% RSLogix 500 project Project2.RSS, saved by version 8.30.00.16 %
PROJECT "UNTITLED"    % processor: Bul.1763 MicroLogix 1100 Series B %

PROGRAM FILES
  LAD 2 "MAIN"  3 rungs
  LAD 3 "IO"  8 rungs
  LAD 4 "CONTROLS"  4 rungs

DATA FILES
  O0 OUTPUT  4 elements
  I1 INPUT  6 elements
  S2 STATUS  66 elements
  B3 BINARY  1 elements
  T4 TIMER  1 elements
  C5 COUNTER  1 elements
  R6 CONTROL  1 elements
  N7 INTEGER  1 elements
  F8 FLOAT  1 elements

LADDER 2 "MAIN"
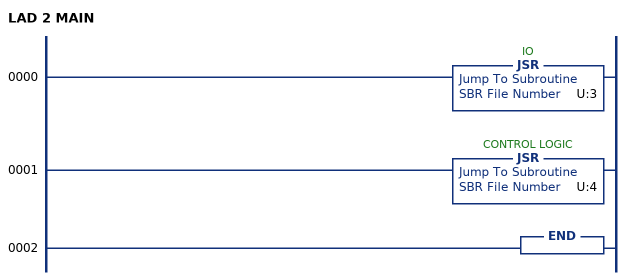
% Rung: 0 %
SOR JSR U:3 EOR
%   U:3  "IO" %
% Rung: 1 %
SOR JSR U:4 EOR
%   U:4  "CONTROL LOGIC" %
% Rung: 2 %
SOR END EOR

LADDER 3 "IO"
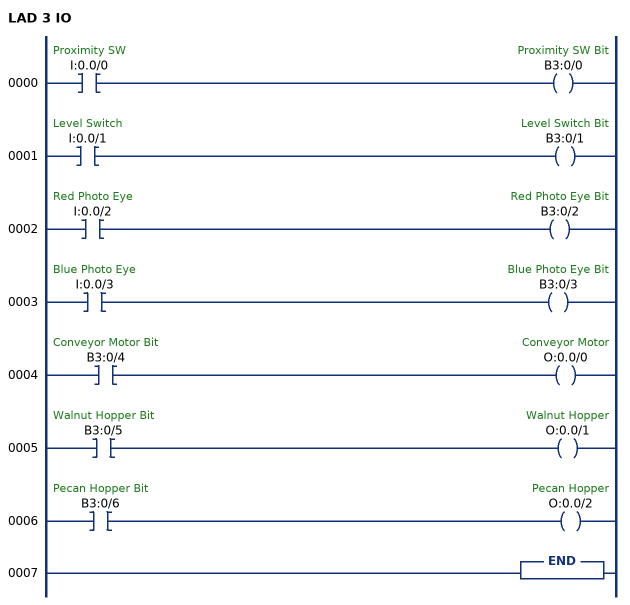
% Rung: 0 %
SOR XIC I:0.0/0 OTE B3:0/0 EOR
%   I:0.0/0  "Proximity SW" %
%   B3:0/0  "Proximity SW Bit" %
% Rung: 1 %
SOR XIC I:0.0/1 OTE B3:0/1 EOR
%   I:0.0/1  "Level Switch" %
%   B3:0/1  "Level Switch Bit" %
% Rung: 2 %
SOR XIC I:0.0/2 OTE B3:0/2 EOR
%   I:0.0/2  "Red Photo Eye" %
%   B3:0/2  "Red Photo Eye Bit" %
% Rung: 3 %
SOR XIC I:0.0/3 OTE B3:0/3 EOR
%   I:0.0/3  "Blue Photo Eye" %
%   B3:0/3  "Blue Photo Eye Bit" %
% Rung: 4 %
SOR XIC B3:0/4 OTE O:0.0/0 EOR
%   B3:0/4  "Conveyor Motor Bit" %
%   O:0.0/0  "Conveyor Motor" %
% Rung: 5 %
SOR XIC B3:0/5 OTE O:0.0/1 EOR
%   B3:0/5  "Walnut Hopper Bit" %
%   O:0.0/1  "Walnut Hopper" %
% Rung: 6 %
SOR XIC B3:0/6 OTE O:0.0/2 EOR
%   B3:0/6  "Pecan Hopper Bit" %
%   O:0.0/2  "Pecan Hopper" %
% Rung: 7 %
SOR END EOR

LADDER 4 "CONTROLS"
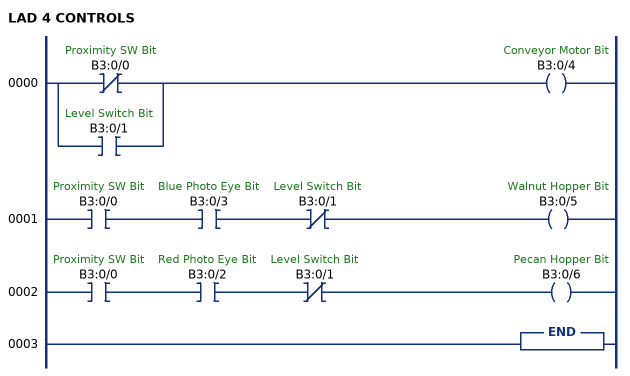
% Rung: 0 %
SOR BST XIO B3:0/0 NXB XIC B3:0/1 BND OTE B3:0/4 EOR
%   B3:0/0  "Proximity SW Bit" %
%   B3:0/1  "Level Switch Bit" %
%   B3:0/4  "Conveyor Motor Bit" %
% Rung: 1 %
SOR XIC B3:0/0 XIC B3:0/3 XIO B3:0/1 OTE B3:0/5 EOR
%   B3:0/0  "Proximity SW Bit" %
%   B3:0/3  "Blue Photo Eye Bit" %
%   B3:0/1  "Level Switch Bit" %
%   B3:0/5  "Walnut Hopper Bit" %
% Rung: 2 %
SOR XIC B3:0/0 XIC B3:0/2 XIO B3:0/1 OTE B3:0/6 EOR
%   B3:0/0  "Proximity SW Bit" %
%   B3:0/2  "Red Photo Eye Bit" %
%   B3:0/1  "Level Switch Bit" %
%   B3:0/6  "Pecan Hopper Bit" %
% Rung: 3 %
SOR END EOR

OTHER DOCUMENTED ADDRESSES
  B3:0/7  FILL_BOX_BIT  "FILL BOX RED LABLE = 1 BLUE LABLE = 0"
